// SIMATIC STEP 7 (V5.x) project TRABAJO DB
// CPU: CPU313 C-2 DP(1)
// station: P_ADR_BUS
// station: Hardware
// station: Equipo SIMATIC 300
// program: Programa S7(1)

SYMBOL_TABLE
"CONTADOR"	FB 201	FB 201	// CONTADOR CON DIFERENCIA DE OPERANDOS
"INTERMITENCIA"	FB 202	FB 202	// INTERMITENCIA CONFIGURABLE
"P MARCHA"	I 0.0	BOOL
"P PARO"	I 0.1	BOOL
"P DESCARGA"	I 0.2	BOOL
"Cycle Execution"	OB 1	OB 1
"MOTOR"	Q 0.0	BOOL
"VAT_1"	VAT 1	
END_SYMBOL_TABLE

FUNCTION_BLOCK "CONTADOR"	// FB 201
TITLE = CONTADOR
//ESTA FUNCION SE ENCARGA DE INCREMENTAR Y DECREMENTAR NUMEROS ENTEROS POSIVOS 
//ENTEROS NEGATIVOS ENTEROS Y COMA FLOTANTE CON PARAMETROS DE INCREMENTO Y 
//DECREMENTO DE ESTERIOR.
//DICHA FUNCION ESTA DCOMPUESTA POR LAS SIGUIENTES ENTRADAS:-UP;VARIABLE BOOLEANO 
//ENCARGADA DE SUMAR LA VARIABLE OPERANDO 1 MAS LA VARIABLE OPERANDO 2 Y MANDAR 
//EL RESULTADO A CONTADOR
//
//-DOWN;VARIABLE BOOLEANO ENCARGADA DE SUMAR LA VARIABLE OPERANDO 1 MAS LA 
//VARIABLE Y MANDAR EL RESULTADO A CONTADOR
//
// 
//-RESET;EL LA ENCARGADA DE PONER A 0 LA VARIABLE CONTADOR.
//-OPERANDO 1 ;VARIABLE TIPO REAL QUE SERA EL PRIMER PARAMETRO DEL CONTADOR.
//-OPERANDO 2 ;;VARIABLE TIPO REAL QUE SERA EL PRIMER PARAMETRO DEL CONTADOR.
//-CONTADOR ;VARIABLE REAL ENCARGADA DE ALMACENAR EL VALOR ACTUAL DEL CONTADOR
//
AUTHOR : JULIAN
FAMILY : PROPIAS
NAME : CONTADPO
VERSION : 1.0
VAR_INPUT
  UP : BOOL ;
  DOWN : BOOL ;
  RESET : BOOL ;
  OPERANDO1 : REAL ;
  OPERANDO2 : REAL ;
END_VAR
VAR_OUTPUT
  CONTADOR : REAL ;
END_VAR
VAR
  FLANCO1 : BOOL ;
  FLANCO2 : BOOL ;
END_VAR
BEGIN
NETWORK
TITLE =
//INCREMENTO DEL CONTADOR
      A     #UP;
      FP    #FLANCO1;
      JNB   _001;
      L     #OPERANDO1;
      L     #OPERANDO2;
      +R;
      T     #CONTADOR;
_001: NOP   0;
NETWORK
TITLE =
//DECREMENTO DEL CONTADOR
      A     #DOWN;
      FP    #FLANCO2;
      JNB   _002;
      L     #OPERANDO1;
      L     #OPERANDO2;
      -R;
      T     #CONTADOR;
_002: NOP   0;
NETWORK
TITLE =
//PUESTA A CERO DEL CONTADOR
      A     #RESET;
      JNB   _003;
      L     0.000000e+00;
      T     #CONTADOR;
_003: NOP   0;
END_FUNCTION_BLOCK

DATA_BLOCK DB 1
AUTHOR : JULIAN
FAMILY : PROPIAS
VERSION : 0.0
"INTERMITENCIA"
BEGIN
END_DATA_BLOCK

DATA_BLOCK DB 2
AUTHOR : JULIAN
FAMILY : PROPIAS
VERSION : 0.0
"CONTADOR"
BEGIN
END_DATA_BLOCK

ORGANIZATION_BLOCK "Cycle Execution"	// OB 1
TITLE = "Main Program Sweep (Cycle)"
VERSION : 0.1
VAR_TEMP
  OB1_EV_CLASS : BYTE ;	//Bits 0-3 = 1 (Coming event), Bits 4-7 = 1 (Event class 1)
  OB1_SCAN_1 : BYTE ;	//1 (Cold restart scan 1 of OB 1), 3 (Scan 2-n of OB 1)
  OB1_PRIORITY : BYTE ;	//Priority of OB Execution
  OB1_OB_NUMBR : BYTE ;	//1 (Organization block 1, OB1)
  OB1_RESERVED_1 : BYTE ;	//Reserved for system
  OB1_RESERVED_2 : BYTE ;	//Reserved for system
  OB1_PREV_CYCLE : INT ;	//Cycle time of previous OB1 scan (milliseconds)
  OB1_MIN_CYCLE : INT ;	//Minimum cycle time of OB1 (milliseconds)
  OB1_MAX_CYCLE : INT ;	//Maximum cycle time of OB1 (milliseconds)
  OB1_DATE_TIME : DATE_AND_TIME ;	//Date and time OB1 started
END_VAR
BEGIN
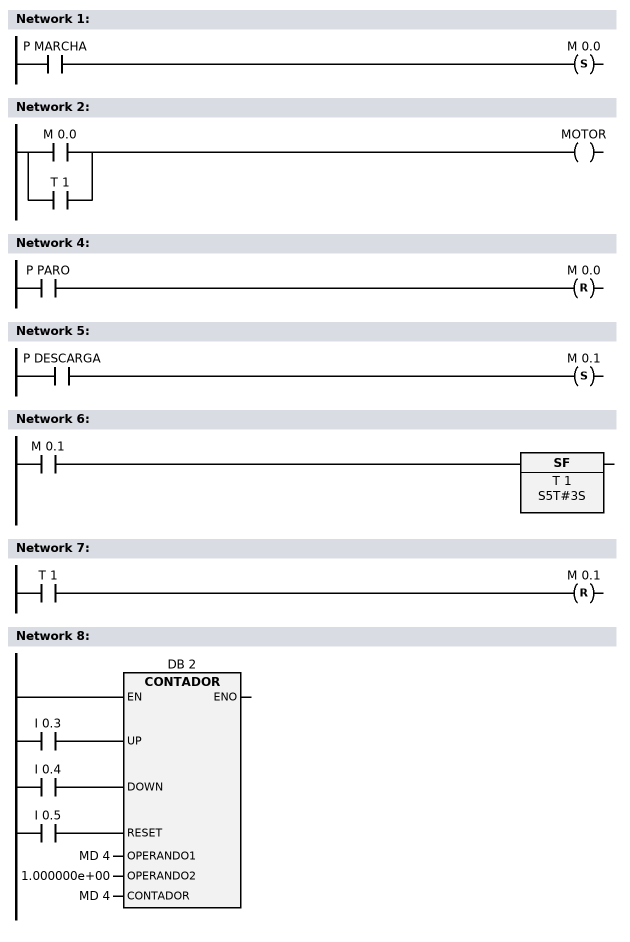
NETWORK
TITLE =
      A     "P MARCHA";
      S     M 0.0;
NETWORK
TITLE =
      O     M 0.0;
      O     T 1;
      =     "MOTOR";
NETWORK
TITLE =
NETWORK
TITLE =
      A     "P PARO";
      R     M 0.0;
NETWORK
TITLE =
      A     "P DESCARGA";
      S     M 0.1;
NETWORK
TITLE =
      A     M 0.1;
      L     S5T#3S;
      SF    T 1;
NETWORK
TITLE =
      A     T 1;
      R     M 0.1;
NETWORK
TITLE =
      A     I 0.3;
      =     L 20.0;
      BLD   103;
      A     I 0.4;
      =     L 20.1;
      BLD   103;
      A     I 0.5;
      =     L 20.2;
      BLD   103;
      CALL  "CONTADOR" , DB 2 (
           UP                       := L 20.0,
           DOWN                     := L 20.1,
           RESET                    := L 20.2,
           OPERANDO1                := MD 4,
           OPERANDO2                := 1.000000e+00,
           CONTADOR                 := MD 4);
      NOP   0;
END_ORGANIZATION_BLOCK
